PROGRAM prgPersistent
VAR
	fbUSV		: FB_WritePersistentData_CX81xx;
	fb_Reboot		: NT_reboot;
	m_Reboot		: BOOL:=FALSE;
END_VAR

fbUSV(
	eSaveModeData:= eUSVSaveMode.eSaveWhenPowerfail, 
	bLoadPersistentDataOk=> , 
	bPowerFailDetect=> , 
	bError=> , 
	bySaveProcess=> , 
	dwStorageLast24h=> , 
	udiErrorCode=> );

	
fb_Reboot(	netid := '',
			delay := 2,
			start := m_Reboot);

END_PROGRAM

(* stored: Version 1.1.0.1, ProductVersion 3.1.4024.12
   POU prgPersistent: Id {ccd67b8a-d866-4216-a145-3575a5a9eafe}, SpecialFunc None *)
